FUNCTION_BLOCK POSTGRES_FETCH
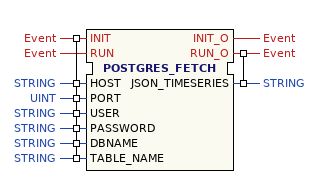
  EVENT_INPUT
    INIT WITH HOST, PORT, USER, PASSWORD, DBNAME, TABLE_NAME;
    RUN;
  END_EVENT
  EVENT_OUTPUT
    INIT_O;
    RUN_O WITH JSON_TIMESERIES;
  END_EVENT
  VAR_INPUT
    HOST : STRING;
    PORT : UINT;
    USER : STRING;
    PASSWORD : STRING;
    DBNAME : STRING;
    TABLE_NAME : STRING;
  END_VAR
  VAR_OUTPUT
    JSON_TIMESERIES : STRING;
  END_VAR
END_FUNCTION_BLOCK
